FUNCTION_BLOCK FB_TelescopeParkedState EXTENDS FB_TelescopeState
VAR_INPUT
END_VAR
VAR_OUTPUT
END_VAR
VAR
END_VAR

IF bInitialize THEN
	pMachine^.State := E_TelescopeState.initializing;
	bInitialize := FALSE;
END_IF

END_FUNCTION_BLOCK

(* stored: Version 1.1.0.1, ProductVersion 3.1.4024.15
   POU FB_TelescopeParkedState: Id {fee317fb-bf48-4714-9d76-2e33fa60c6a5}, SpecialFunc None *)
